# EPICS autosave request: stdApp/Db/IK320card_settings.req
# FILE... IK320card_settings.req
# USAGE.. IK320card.db fields autosave'd.
$(P)IK320:$(sw2)$(axis).B
$(P)IK320:$(sw2)$(axis)direction.VAL
$(P)IK320:$(sw2)$(axis)raw.DESC
$(P)IK320:$(sw2)$(axis)raw.EGU
$(P)IK320:$(sw2)$(axis)raw.ASLO
$(P)IK320:$(sw2)$(axis)prec.VAL
